// TIA Portal project "OPCUA_V16" (V16)

(* hardware
DEVICE "S7-1200-Station_1"  S7-1200 Station
   slot 0: "Baugruppenträger_0"  S7-1200 Rack  Rack  V1.0
   slot 1: "PLC_1"  CPU 1215C AC/DC/Rly  6ES7 215-1BG40-0XB0  V4.2
   slot 2: "AI 4x13BIT_1"  6ES7 231-4HD32-0XB0  V2.0
DEVICE "S71500/ET200MP-Station_2"  S7-1500 station
   slot 0: "Profilschiene_0"  Rack  6ES7 590-1***0-0AA0
   slot 1: "PLC_2"  CPU 1511-1 PN  6ES7 511-1AK02-0AB0  V2.8
      slot 3: "CPU-Display_1"  6ES7591-1AA00-0AA0
      slot 32768: "PROFINET-Schnittstelle_1"  X1
      slot 34817: "Virtual CP interface port_1"  Virtual CP interface port  Virtual CP interface port
*)

// ===== PLC "PLC_1"  CPU 1215C AC/DC/Rly =====

// folder: IOTDataCollect

DATA_BLOCK "IOT_Data"   // DB1
{ S7_Optimized_Access := 'TRUE' }
VERSION : 0.1
   VAR
      IOT_Bool : Bool;
      IOT_Int : Int;
      IOT_Real : Real;
   END_VAR
BEGIN
END_DATA_BLOCK

DATA_BLOCK "instIOTDataGenerator"   // DB2
{ S7_Optimized_Access := 'TRUE' }
VERSION : 0.1
// stored: InstanceOfName IOTDataGenerator
"IOTDataGenerator"
BEGIN
END_DATA_BLOCK

DATA_BLOCK "IOT_DataClassic"   // DB3
{ S7_Optimized_Access := 'FALSE' }
VERSION : 0.1
   VAR
      IOT_Bool : Bool;
      IOT_Int : Int;
      IOT_Real : Real;
   END_VAR
BEGIN
END_DATA_BLOCK

DATA_BLOCK "HoldingRegisterRead"   // DB4
{ S7_Optimized_Access := 'TRUE' }
VERSION : 0.1
   VAR
      holdingRegister : Array[0..65535] of Word;
   END_VAR
BEGIN
END_DATA_BLOCK

DATA_BLOCK "instMobdusServer"   // DB6
{ S7_Optimized_Access := 'TRUE' }
VERSION : 0.1
// stored: InstanceOfName MobdusServer
"MobdusServer"
BEGIN
END_DATA_BLOCK

DATA_BLOCK "ModbusData"   // DB100
{ S7_Optimized_Access := 'TRUE' }
VERSION : 0.1
   VAR
      connectParamServer : TCON_IP_v4;
      serverData : Struct
         disconnect : Bool;
         ndr : Bool;
         dataRead : Bool;
         error : Bool;
         status : Word;
         statusSave : Word;
      END_STRUCT;
      holdingRegister : Array[0..65535] of Word;
   END_VAR
BEGIN
   connectParamServer.InterfaceId := 64;
   connectParamServer.ID := 2;
   connectParamServer.ConnectionType := 11;
   connectParamServer.ActiveEstablished := 0;
   connectParamServer.RemoteAddress.ADDR[1] := 0;
   connectParamServer.RemoteAddress.ADDR[2] := 0;
   connectParamServer.RemoteAddress.ADDR[3] := 0;
   connectParamServer.RemoteAddress.ADDR[4] := 0;
   connectParamServer.RemotePort := 0;
   connectParamServer.LocalPort := 503;
END_DATA_BLOCK

FUNCTION_BLOCK "IOTDataGenerator"   // FB1, SCL
{ S7_Optimized_Access := 'TRUE' }
VERSION : 0.1
   VAR_OUTPUT
      SinusValue : Real;
      RandomInt : Int;
      IOT_Bool : Bool;
      IOT_Time : Time;
   END_VAR
   VAR
      angle : Real;
   END_VAR
   VAR_TEMP
      SystemTime : DTL;
      diTime : DInt;
      rTime : Real;
      rRandom : Real;
      RDTimeRetValue : Int;
      toDay : Time_Of_Day;
   END_VAR
   VAR CONSTANT
      pi : Real := 3.141593;
      SinusStep : Real := 0.02;
      SinusAmplitude : Real := 1.0;
      RandomMax : Int := 32767;
   END_VAR
BEGIN
   //FB IOTDataGenerator : Fuction Block to Generate some values 

   // Sinus
   IF #angle > 2 * #pi THEN
       #angle := 0;
   END_IF;

   #SinusValue := #SinusAmplitude * SIN(#angle);
   #angle := #angle + #SinusStep;

   #RDTimeRetValue :=  RD_SYS_T(#SystemTime);
   //Random Integer


   // calculate random number
   #toDay := DTL_TO_TOD(#SystemTime);
   #diTime := TOD_TO_DINT(#toDay);
   #rTime := DINT_TO_REAL(#diTime);
   #rRandom := SIN(#rTime);
   #RandomInt := REAL_TO_INT(#rRandom * #RandomMax);

   //Bool
   //
   #IOT_Bool := (#RandomInt > 0);

   //Time
   //
   #IOT_Time := #toDay;
END_FUNCTION_BLOCK

FUNCTION_BLOCK "MobdusServer"   // FB2, SCL
{ S7_Optimized_Access := 'TRUE' }
VERSION : 0.1
   VAR_INPUT
      disconnect : Bool;
   END_VAR
   VAR_OUTPUT
      ndr : Bool;
      dataRead : Bool;
      error : Bool;
      status : Word;
   END_VAR
   VAR_IN_OUT
      dataBuffer : Variant;
      connectParamServer : Variant;
   END_VAR
   VAR
      instModbusServer : MB_SERVER;
   END_VAR
BEGIN
   #instModbusServer(DISCONNECT:=#disconnect,
                     NDR=>#ndr,
                     DR=>#dataRead,
                     ERROR=>#error,
                     STATUS=>#status,
                     MB_HOLD_REG:=#dataBuffer,
                     CONNECT:=#connectParamServer);
END_FUNCTION_BLOCK

FUNCTION "SetHoldingRegisterData" : Void   // FC1, SCL
{ S7_Optimized_Access := 'TRUE' }
VERSION : 0.1
   VAR_TEMP
      tmprealdw : DWord;
   END_VAR
BEGIN

   #tmprealdw := REAL_TO_DWORD("IOT_Data".IOT_Real);


   "ModbusData".holdingRegister[0] := BOOL_TO_WORD("IOT_Data".IOT_Bool);
   "ModbusData".holdingRegister[1] := INT_TO_WORD("IOT_Data".IOT_Int);
   "ModbusData".holdingRegister[2] := #tmprealdw AND 16#0000FFFF;
   "ModbusData".holdingRegister[3] := SHR(IN := #tmprealdw, N := 16) AND 16#0000FFFF;
END_FUNCTION

ORGANIZATION_BLOCK "Main"   // OB1, FBD, ProgramCycle
TITLE = "Main Program Sweep (Cycle)"
{ S7_Optimized_Access := 'TRUE' }
VERSION : 0.1
   VAR_INPUT
      Initial_Call : Bool;   // Initial call of this OB
      Remanence : Bool;   // =True, if remanent data are available
   END_VAR
   VAR_TEMP   // added for the SCL form of the ladder/FBD networks
      _w1 : Bool;
   END_VAR
BEGIN

REGION Network 1
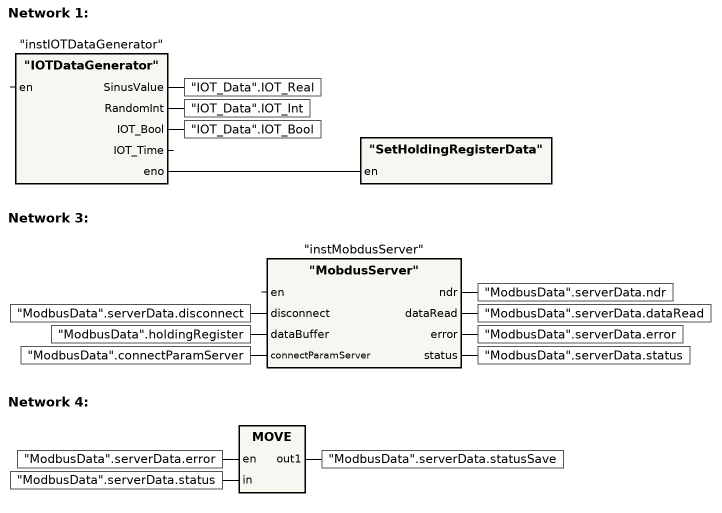
   "instIOTDataGenerator"(SinusValue => "IOT_Data".IOT_Real,   // "IOTDataGenerator"
                          RandomInt => "IOT_Data".IOT_Int,
                          IOT_Bool => "IOT_Data".IOT_Bool,
                          ENO => #_w1);
   IF #_w1 THEN "SetHoldingRegisterData"(); END_IF;
END_REGION

REGION Network 2 (SCL)
   "IOT_DataClassic".IOT_Real := "IOT_Data".IOT_Real;
   "IOT_DataClassic".IOT_Int := "IOT_Data".IOT_Int;
   "IOT_DataClassic".IOT_Bool := "IOT_Data".IOT_Bool;
END_REGION

REGION Network 3
   "instMobdusServer"(disconnect := "ModbusData".serverData.disconnect,   // "MobdusServer"
                      dataBuffer := "ModbusData".holdingRegister,
                      connectParamServer := "ModbusData".connectParamServer,
                      ndr => "ModbusData".serverData.ndr,
                      dataRead => "ModbusData".serverData.dataRead,
                      error => "ModbusData".serverData.error,
                      status => "ModbusData".serverData.status);
END_REGION

REGION Network 4
   IF "ModbusData".serverData.error THEN
       "ModbusData".serverData.statusSave := "ModbusData".serverData.status;
   END_IF;
END_REGION
END_ORGANIZATION_BLOCK

// ===== PLC "PLC_2"  CPU 1511-1 PN =====

TYPE "IOT_DataType"
   STRUCT
      IOT_Bool : Bool;
      IOT_Int : Int;
      IOT_Real : Real;
      IOT_Time : Time;
   END_STRUCT;
END_TYPE

// folder: IOTDataCollect

DATA_BLOCK "IOT_Data"   // DB1
{ S7_Optimized_Access := 'TRUE' }
VERSION : 0.1
   VAR
      IOT_Bool : Bool;
      IOT_Int : Int;
      IOT_Real : Real;
   END_VAR
BEGIN
END_DATA_BLOCK

DATA_BLOCK "instIOTDataGenerator"   // DB2
{ S7_Optimized_Access := 'TRUE' }
VERSION : 0.1
// stored: InstanceOfName IOTDataGenerator
"IOTDataGenerator"
BEGIN
END_DATA_BLOCK

DATA_BLOCK "IOT_DataClassic"   // DB3
{ S7_Optimized_Access := 'FALSE' }
VERSION : 0.1
   VAR
      IOT_Bool : Bool;
      IOT_Int : Int;
      IOT_Real : Real;
   END_VAR
BEGIN
END_DATA_BLOCK

DATA_BLOCK "HoldingRegisterRead"   // DB4
{ S7_Optimized_Access := 'TRUE' }
VERSION : 0.1
   VAR
      holdingRegister : Array[0..65535] of Word;
   END_VAR
BEGIN
END_DATA_BLOCK

DATA_BLOCK "instMobdusServer"   // DB6
{ S7_Optimized_Access := 'TRUE' }
VERSION : 0.1
// stored: InstanceOfName MobdusServer
"MobdusServer"
BEGIN
END_DATA_BLOCK

DATA_BLOCK "ModbusData"   // DB100
{ S7_Optimized_Access := 'TRUE' }
VERSION : 0.1
   VAR
      connectParamServer : TCON_IP_v4;
      serverData : Struct
         disconnect : Bool;
         ndr : Bool;
         dataRead : Bool;
         error : Bool;
         status : Word;
         statusSave : Word;
      END_STRUCT;
      holdingRegister : Array[0..65535] of Word;
   END_VAR
BEGIN
   connectParamServer.InterfaceId := 64;
   connectParamServer.ID := 2;
   connectParamServer.ConnectionType := 11;
   connectParamServer.ActiveEstablished := 0;
   connectParamServer.RemoteAddress.ADDR[1] := 0;
   connectParamServer.RemoteAddress.ADDR[2] := 0;
   connectParamServer.RemoteAddress.ADDR[3] := 0;
   connectParamServer.RemoteAddress.ADDR[4] := 0;
   connectParamServer.RemotePort := 0;
   connectParamServer.LocalPort := 503;
END_DATA_BLOCK

FUNCTION_BLOCK "IOTDataGenerator"   // FB1, SCL
{ S7_Optimized_Access := 'TRUE' }
VERSION : 0.1
   VAR_OUTPUT
      SinusValue : Real;
      RandomInt : Int;
      IOT_Bool : Bool;
   END_VAR
   VAR
      angle : Real;
   END_VAR
   VAR_TEMP
      SystemTime : Time;
      diTime : DInt;
      rTime : Real;
      rRandom : Real;
   END_VAR
   VAR CONSTANT
      pi : Real := 3.141593;
      SinusStep : Real := 0.02;
      SinusAmplitude : Real := 1.0;
      RandomMax : Int := 32767;
   END_VAR
BEGIN
   //FB IOTDataGenerator : Fuction Block to Generate some values 

   // Sinus
   IF #angle > 2 * #pi THEN
       #angle := 0;
   END_IF;

   #SinusValue := #SinusAmplitude * SIN(#angle);
   #angle := #angle + #SinusStep;

   //Random Integer
   #SystemTime := TIME_TCK();

   // calculate random number
   #diTime := TIME_TO_DINT(#SystemTime);
   #rTime := DINT_TO_REAL(#diTime);
   #rRandom := SIN(#rTime);
   #RandomInt := REAL_TO_INT(#rRandom * #RandomMax);

   //Bool
   //
   #IOT_Bool := (#RandomInt > 0);
END_FUNCTION_BLOCK

FUNCTION_BLOCK "MobdusServer"   // FB2, SCL
{ S7_Optimized_Access := 'TRUE' }
VERSION : 0.1
   VAR_INPUT
      disconnect : Bool;
   END_VAR
   VAR_OUTPUT
      ndr : Bool;
      dataRead : Bool;
      error : Bool;
      status : Word;
   END_VAR
   VAR_IN_OUT
      dataBuffer : Variant;
      connectParamServer : Variant;
   END_VAR
   VAR
      instModbusServer : MB_SERVER;
   END_VAR
BEGIN
   #instModbusServer(DISCONNECT:=#disconnect,
                     NDR=>#ndr,
                     DR=>#dataRead,
                     ERROR=>#error,
                     STATUS=>#status,
                     MB_HOLD_REG:=#dataBuffer,
                     CONNECT:=#connectParamServer);
END_FUNCTION_BLOCK

FUNCTION "SetHoldingRegisterData" : Void   // FC1, SCL
{ S7_Optimized_Access := 'TRUE' }
VERSION : 0.1
   VAR_TEMP
      tmprealdw : DWord;
   END_VAR
BEGIN

   #tmprealdw := REAL_TO_DWORD("IOT_Data".IOT_Real);


   "ModbusData".holdingRegister[0] := BOOL_TO_WORD("IOT_Data".IOT_Bool);
   "ModbusData".holdingRegister[1] := INT_TO_WORD("IOT_Data".IOT_Int);
   "ModbusData".holdingRegister[2] := #tmprealdw AND 16#0000FFFF;
   "ModbusData".holdingRegister[3] := SHR(IN := #tmprealdw, N := 16) AND 16#0000FFFF;
END_FUNCTION

ORGANIZATION_BLOCK "Main"   // OB1, FBD, ProgramCycle
TITLE = "Main Program Sweep (Cycle)"
{ S7_Optimized_Access := 'TRUE' }
VERSION : 0.1
   VAR_INPUT
      Initial_Call : Bool;   // Initial call of this OB
      Remanence : Bool;   // =True, if remanent data are available
   END_VAR
   VAR_TEMP   // added for the SCL form of the ladder/FBD networks
      _w1 : Bool;
   END_VAR
BEGIN

REGION Network 1
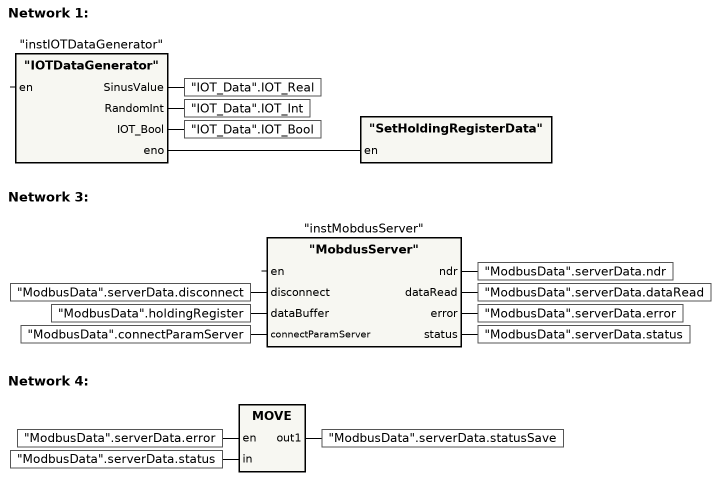
   "instIOTDataGenerator"(SinusValue => "IOT_Data".IOT_Real,   // "IOTDataGenerator"
                          RandomInt => "IOT_Data".IOT_Int,
                          IOT_Bool => "IOT_Data".IOT_Bool,
                          ENO => #_w1);
   IF #_w1 THEN "SetHoldingRegisterData"(); END_IF;
END_REGION

REGION Network 2 (SCL)
   "IOT_DataClassic".IOT_Real := "IOT_Data".IOT_Real;
   "IOT_DataClassic".IOT_Int := "IOT_Data".IOT_Int;
   "IOT_DataClassic".IOT_Bool := "IOT_Data".IOT_Bool;
END_REGION

REGION Network 3
   "instMobdusServer"(disconnect := "ModbusData".serverData.disconnect,   // "MobdusServer"
                      dataBuffer := "ModbusData".holdingRegister,
                      connectParamServer := "ModbusData".connectParamServer,
                      ndr => "ModbusData".serverData.ndr,
                      dataRead => "ModbusData".serverData.dataRead,
                      error => "ModbusData".serverData.error,
                      status => "ModbusData".serverData.status);
END_REGION

REGION Network 4
   IF "ModbusData".serverData.error THEN
       "ModbusData".serverData.statusSave := "ModbusData".serverData.status;
   END_IF;
END_REGION
END_ORGANIZATION_BLOCK